SUBAPPLICATION Uebung_060_sub_Outputs (* für TC-SC also Task Controller Section Control *)
  (* Standard: 61499-2; Description: Copyright (c) 2024 Meisterschulen am Ostbahnhof This program and the accompanying materials are made available under the terms of the Eclipse Public License 2.0 which is available at https://www.eclipse.org/legal/epl-2.0/ SPDX-License-Identifier: EPL-2.0 *)
  (* Version 1.0, 2024-02-29, Franz Höpfinger, Meisterschulen am Ostbahnhof *)
  PACKAGE Uebungen;
  IMPORT logiBUS::io::DQ::logiBUS_DO::Output_Q1;
  IMPORT logiBUS::io::DQ::logiBUS_DO::Output_Q2;
  IMPORT logiBUS::io::DQ::logiBUS_DO::Output_Q3;
  IMPORT logiBUS::io::DQ::logiBUS_DO::Output_Q4;
  IMPORT logiBUS::io::DQ::logiBUS_DO::Output_Q5;
  IMPORT logiBUS::io::DQ::logiBUS_DO::Output_Q6;
  IMPORT logiBUS::io::DQ::logiBUS_DO::Output_Q7;
  IMPORT logiBUS::io::DQ::logiBUS_DO::Output_Q8;
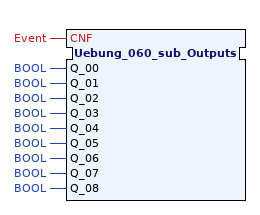
  EVENT_INPUT
    CNF;
  END_EVENT
  VAR_INPUT
    Q_00 : BOOL;
    Q_01 : BOOL;
    Q_02 : BOOL;
    Q_03 : BOOL;
    Q_04 : BOOL;
    Q_05 : BOOL;
    Q_06 : BOOL;
    Q_07 : BOOL;
    Q_08 : BOOL;
  END_VAR
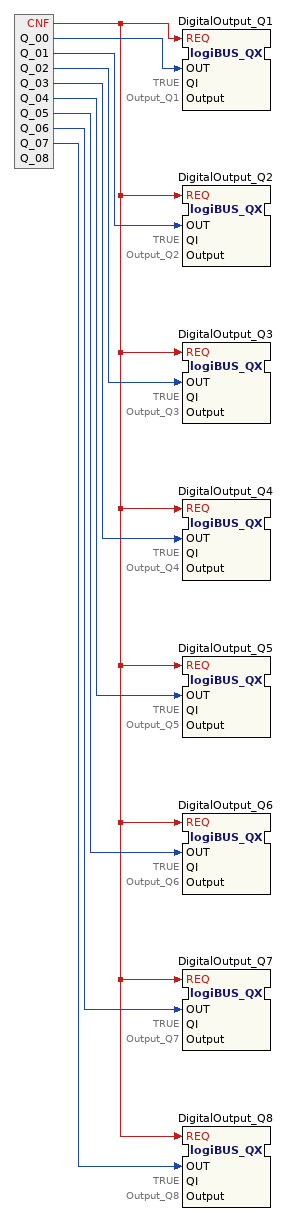
  FBS
    DigitalOutput_Q4 : logiBUS::io::DQ::logiBUS_QX(QI := TRUE, Output := Output_Q4);
    DigitalOutput_Q7 : logiBUS::io::DQ::logiBUS_QX(QI := TRUE, Output := Output_Q7);
    DigitalOutput_Q1 : logiBUS::io::DQ::logiBUS_QX(QI := TRUE, Output := Output_Q1);
    DigitalOutput_Q5 : logiBUS::io::DQ::logiBUS_QX(QI := TRUE, Output := Output_Q5);
    DigitalOutput_Q2 : logiBUS::io::DQ::logiBUS_QX(QI := TRUE, Output := Output_Q2);
    DigitalOutput_Q6 : logiBUS::io::DQ::logiBUS_QX(QI := TRUE, Output := Output_Q6);
    DigitalOutput_Q8 : logiBUS::io::DQ::logiBUS_QX(QI := TRUE, Output := Output_Q8);
    DigitalOutput_Q3 : logiBUS::io::DQ::logiBUS_QX(QI := TRUE, Output := Output_Q3);
  END_FBS
  EVENT_CONNECTIONS
    CNF TO DigitalOutput_Q4.REQ;
    CNF TO DigitalOutput_Q7.REQ;
    CNF TO DigitalOutput_Q1.REQ;
    CNF TO DigitalOutput_Q5.REQ;
    CNF TO DigitalOutput_Q2.REQ;
    CNF TO DigitalOutput_Q6.REQ;
    CNF TO DigitalOutput_Q8.REQ;
    CNF TO DigitalOutput_Q3.REQ;
  END_CONNECTIONS
  DATA_CONNECTIONS
    Q_06 TO DigitalOutput_Q7.OUT;
    Q_00 TO DigitalOutput_Q1.OUT;
    Q_04 TO DigitalOutput_Q5.OUT;
    Q_01 TO DigitalOutput_Q2.OUT;
    Q_05 TO DigitalOutput_Q6.OUT;
    Q_02 TO DigitalOutput_Q3.OUT;
    Q_03 TO DigitalOutput_Q4.OUT;
    Q_07 TO DigitalOutput_Q8.OUT;
  END_CONNECTIONS
END_SUBAPPLICATION
